TYPE Weld_Robot :
STRUCT
	i_Home 		: BOOL;
	i_Prg_No	: INT;
	i_Start		: BOOL;	
	i_Area_Ok	: BOOL;
	
	o_Weld_Comp	: BOOL;
	
END_STRUCT
END_TYPE

(* stored: Version 1.1.0.1, ProductVersion 3.1.4024.16
   DUT Weld_Robot: Id {fa3c1610-845c-43f1-ba63-5a5e0098c2d5} *)
